# EPICS substitutions: db/Beckhoff_5XXX/ecmcEL5101.substitutions
# All fields related to postion scaling and alarms
file "ecmcEcSlave.template"
{
  pattern {}
          {}
}

file "ecmcEL5101-chX.template"
{
    pattern {CH_ID}
            {01   }

}
